# EPICS substitutions: iocBoot/iocgalil/galil_digital_ports.substitutions
# Description:
# digital/binary port substitution file.
#
# This library is free software; you can redistribute it and/or
# modify it under the terms of the GNU Lesser General Public
# Licence as published by the Free Software Foundation; either
# version 2.1 of the Licence, or (at your option) any later version.
#
# This library is distributed in the hope that it will be useful,
# but WITHOUT ANY WARRANTY; without even the implied warranty of
# MERCHANTABILITY or FITNESS FOR A PARTICULAR PURPOSE.  See the GNU
# Lesser General Public Licence for more details.
#
# You should have received a copy of the GNU Lesser General Public
# Licence along with this library; if not, write to the Free Software
# Foundation, Inc., 51 Franklin St, Fifth Floor, Boston, MA 02110-1301 USA.
#
# Contact details:
# mark.clift@synchrotron.org.au
# 800 Blackburn Road, Clayton, Victoria 3168, Australia.
#

# P    - PV prefix
# R    - Record Name
# PORT - Asyn port name
# BYTE - Hardware byte to read
# MASK - Mask for this bit

# Digital IO naming
# $(P)$(R)<Byte or word num><Type Bo or Bi><Bit>

file "$(TOP)/db/galil_digital_in_bit.template"
{
pattern {P,      R,          PORT,  BYTE,  MASK,     ZNAM,  ONAM,  ZSV,        OSV         }

# DMC = Digital motor controller
# DMC binary inputs are organized in bytes
	{CEL:GALIL,  Galil0Bi0,  Galil, 0,     0x000001, "Off", "On",  "NO_ALARM", "NO_ALARM"  }
	{CEL:GALIL,  Galil0Bi1,  Galil, 0,     0x000002, "Off", "On",  "NO_ALARM", "NO_ALARM"  }
	{CEL:GALIL,  Galil0Bi2,  Galil, 0,     0x000004, "Off", "On",  "NO_ALARM", "NO_ALARM"  }
	{CEL:GALIL,  Galil0Bi3,  Galil, 0,     0x000008, "Off", "On",  "NO_ALARM", "NO_ALARM"  }
	{CEL:GALIL,  Galil0Bi4,  Galil, 0,     0x000010, "Off", "On",  "NO_ALARM", "NO_ALARM"  }
	{CEL:GALIL,  Galil0Bi5,  Galil, 0,     0x000020, "Off", "On",  "NO_ALARM", "NO_ALARM"  }
	{CEL:GALIL,  Galil0Bi6,  Galil, 0,     0x000040, "Off", "On",  "NO_ALARM", "NO_ALARM"  }
	{CEL:GALIL,  Galil0Bi7,  Galil, 0,     0x000080, "Off", "On",  "NO_ALARM", "NO_ALARM"  }

	{CEL:GALIL,  Galil1Bi0,  Galil, 1,     0x000001, "Off", "On",  "NO_ALARM", "NO_ALARM"  }
	{CEL:GALIL,  Galil1Bi1,  Galil, 1,     0x000002, "Off", "On",  "NO_ALARM", "NO_ALARM"  }
	{CEL:GALIL,  Galil1Bi2,  Galil, 1,     0x000004, "Off", "On",  "NO_ALARM", "NO_ALARM"  }
	{CEL:GALIL,  Galil1Bi3,  Galil, 1,     0x000008, "Off", "On",  "NO_ALARM", "NO_ALARM"  }
	{CEL:GALIL,  Galil1Bi4,  Galil, 1,     0x000010, "Off", "On",  "NO_ALARM", "NO_ALARM"  }
	{CEL:GALIL,  Galil1Bi5,  Galil, 1,     0x000020, "Off", "On",  "NO_ALARM", "NO_ALARM"  }
	{CEL:GALIL,  Galil1Bi6,  Galil, 1,     0x000040, "Off", "On",  "NO_ALARM", "NO_ALARM"  }
	{CEL:GALIL,  Galil1Bi7,  Galil, 1,     0x000080, "Off", "On",  "NO_ALARM", "NO_ALARM"  }

	{CEL:GALIL,  Galil2Bi0,  Galil, 2,     0x000001, "Off", "On",  "NO_ALARM", "NO_ALARM"  }
	{CEL:GALIL,  Galil2Bi1,  Galil, 2,     0x000002, "Off", "On",  "NO_ALARM", "NO_ALARM"  }
	{CEL:GALIL,  Galil2Bi2,  Galil, 2,     0x000004, "Off", "On",  "NO_ALARM", "NO_ALARM"  }
	{CEL:GALIL,  Galil2Bi3,  Galil, 2,     0x000008, "Off", "On",  "NO_ALARM", "NO_ALARM"  }
	{CEL:GALIL,  Galil2Bi4,  Galil, 2,     0x000010, "Off", "On",  "NO_ALARM", "NO_ALARM"  }
	{CEL:GALIL,  Galil2Bi5,  Galil, 2,     0x000020, "Off", "On",  "NO_ALARM", "NO_ALARM"  }
	{CEL:GALIL,  Galil2Bi6,  Galil, 2,     0x000040, "Off", "On",  "NO_ALARM", "NO_ALARM"  }
	{CEL:GALIL,  Galil2Bi7,  Galil, 2,     0x000080, "Off", "On",  "NO_ALARM", "NO_ALARM"  }

# RIO binary inputs are organized in bytes
	{RIO01,  Galil0Bi0,  RIO,   0,     0x000001, "Off", "On",  "NO_ALARM", "NO_ALARM"  }
	{RIO01,  Galil0Bi1,  RIO,   0,     0x000002, "Off", "On",  "NO_ALARM", "NO_ALARM"  }
	{RIO01,  Galil0Bi2,  RIO,   0,     0x000004, "Off", "On",  "NO_ALARM", "NO_ALARM"  }
	{RIO01,  Galil0Bi3,  RIO,   0,     0x000008, "Off", "On",  "NO_ALARM", "NO_ALARM"  }
	{RIO01,  Galil0Bi4,  RIO,   0,     0x000010, "Off", "On",  "NO_ALARM", "NO_ALARM"  }
	{RIO01,  Galil0Bi5,  RIO,   0,     0x000020, "Off", "On",  "NO_ALARM", "NO_ALARM"  }
	{RIO01,  Galil0Bi6,  RIO,   0,     0x000040, "Off", "On",  "NO_ALARM", "NO_ALARM"  }
	{RIO01,  Galil0Bi7,  RIO,   0,     0x000080, "Off", "On",  "NO_ALARM", "NO_ALARM"  }

	{RIO01,  Galil1Bi0,  RIO,   1,     0x000001, "Off", "On",  "NO_ALARM", "NO_ALARM"  }
	{RIO01,  Galil1Bi1,  RIO,   1,     0x000002, "Off", "On",  "NO_ALARM", "NO_ALARM"  }
	{RIO01,  Galil1Bi2,  RIO,   1,     0x000004, "Off", "On",  "NO_ALARM", "NO_ALARM"  }
	{RIO01,  Galil1Bi3,  RIO,   1,     0x000008, "Off", "On",  "NO_ALARM", "NO_ALARM"  }
	{RIO01,  Galil1Bi4,  RIO,   1,     0x000010, "Off", "On",  "NO_ALARM", "NO_ALARM"  }
	{RIO01,  Galil1Bi5,  RIO,   1,     0x000020, "Off", "On",  "NO_ALARM", "NO_ALARM"  }
	{RIO01,  Galil1Bi6,  RIO,   1,     0x000040, "Off", "On",  "NO_ALARM", "NO_ALARM"  }
	{RIO01,  Galil1Bi7,  RIO,   1,     0x000080, "Off", "On",  "NO_ALARM", "NO_ALARM"  }

	{RIO01,  Galil2Bi0,  RIO,   2,     0x000001, "Off", "On",  "NO_ALARM", "NO_ALARM"  }
	{RIO01,  Galil2Bi1,  RIO,   2,     0x000002, "Off", "On",  "NO_ALARM", "NO_ALARM"  }
	{RIO01,  Galil2Bi2,  RIO,   2,     0x000004, "Off", "On",  "NO_ALARM", "NO_ALARM"  }
	{RIO01,  Galil2Bi3,  RIO,   2,     0x000008, "Off", "On",  "NO_ALARM", "NO_ALARM"  }
	{RIO01,  Galil2Bi4,  RIO,   2,     0x000010, "Off", "On",  "NO_ALARM", "NO_ALARM"  }
	{RIO01,  Galil2Bi5,  RIO,   2,     0x000020, "Off", "On",  "NO_ALARM", "NO_ALARM"  }
	{RIO01,  Galil2Bi6,  RIO,   2,     0x000040, "Off", "On",  "NO_ALARM", "NO_ALARM"  }
	{RIO01,  Galil2Bi7,  RIO,   2,     0x000080, "Off", "On",  "NO_ALARM", "NO_ALARM"  }

}

# P    - PV prefix
# R    - Record Name
# PORT - Asyn port name
# WORD - Hardware word to read
# MASK - Mask for this bit

file "$(TOP)/db/galil_digital_out_bit.template"
{
pattern {P,      R,           PORT,  WORD,  MASK,     ZNAM,  ONAM,  ZSV,        OSV         }

# DMC binary outputs are organized in 16bit words
	{CEL:GALIL,  Galil0Bo0,   Galil, 0,     0x000001, "Off", "On",  "NO_ALARM", "NO_ALARM"  }
	{CEL:GALIL,  Galil0Bo1,   Galil, 0,     0x000002, "Off", "On",  "NO_ALARM", "NO_ALARM"  }
	{CEL:GALIL,  Galil0Bo2,   Galil, 0,     0x000004, "Off", "On",  "NO_ALARM", "NO_ALARM"  }
	{CEL:GALIL,  Galil0Bo3,   Galil, 0,     0x000008, "Off", "On",  "NO_ALARM", "NO_ALARM"  }
	{CEL:GALIL,  Galil0Bo4,   Galil, 0,     0x000010, "Off", "On",  "NO_ALARM", "NO_ALARM"  }
	{CEL:GALIL,  Galil0Bo5,   Galil, 0,     0x000020, "Off", "On",  "NO_ALARM", "NO_ALARM"  }
	{CEL:GALIL,  Galil0Bo6,   Galil, 0,     0x000040, "Off", "On",  "NO_ALARM", "NO_ALARM"  }
	{CEL:GALIL,  Galil0Bo7,   Galil, 0,     0x000080, "Off", "On",  "NO_ALARM", "NO_ALARM"  }
	{CEL:GALIL,  Galil0Bo8,   Galil, 0,     0x000100, "Off", "On",  "NO_ALARM", "NO_ALARM"  }
	{CEL:GALIL,  Galil0Bo9,   Galil, 0,     0x000200, "Off", "On",  "NO_ALARM", "NO_ALARM"  }
	{CEL:GALIL,  Galil0Bo10,  Galil, 0,     0x000400, "Off", "On",  "NO_ALARM", "NO_ALARM"  }
	{CEL:GALIL,  Galil0Bo11,  Galil, 0,     0x000800, "Off", "On",  "NO_ALARM", "NO_ALARM"  }
	{CEL:GALIL,  Galil0Bo12,  Galil, 0,     0x001000, "Off", "On",  "NO_ALARM", "NO_ALARM"  }
	{CEL:GALIL,  Galil0Bo13,  Galil, 0,     0x002000, "Off", "On",  "NO_ALARM", "NO_ALARM"  }
	{CEL:GALIL,  Galil0Bo14,  Galil, 0,     0x004000, "Off", "On",  "NO_ALARM", "NO_ALARM"  }
	{CEL:GALIL,  Galil0Bo15,  Galil, 0,     0x008000, "Off", "On",  "NO_ALARM", "NO_ALARM"  }

	{CEL:GALIL,  Galil1Bo0,   Galil, 1,     0x000001, "Off", "On",  "NO_ALARM", "NO_ALARM"  }
	{CEL:GALIL,  Galil1Bo1,   Galil, 1,     0x000002, "Off", "On",  "NO_ALARM", "NO_ALARM"  }
	{CEL:GALIL,  Galil1Bo2,   Galil, 1,     0x000004, "Off", "On",  "NO_ALARM", "NO_ALARM"  }
	{CEL:GALIL,  Galil1Bo3,   Galil, 1,     0x000008, "Off", "On",  "NO_ALARM", "NO_ALARM"  }
	{CEL:GALIL,  Galil1Bo4,   Galil, 1,     0x000010, "Off", "On",  "NO_ALARM", "NO_ALARM"  }
	{CEL:GALIL,  Galil1Bo5,   Galil, 1,     0x000020, "Off", "On",  "NO_ALARM", "NO_ALARM"  }
	{CEL:GALIL,  Galil1Bo6,   Galil, 1,     0x000040, "Off", "On",  "NO_ALARM", "NO_ALARM"  }
	{CEL:GALIL,  Galil1Bo7,   Galil, 1,     0x000080, "Off", "On",  "NO_ALARM", "NO_ALARM"  }
	{CEL:GALIL,  Galil1Bo8,   Galil, 1,     0x000100, "Off", "On",  "NO_ALARM", "NO_ALARM"  }
	{CEL:GALIL,  Galil1Bo9,   Galil, 1,     0x000200, "Off", "On",  "NO_ALARM", "NO_ALARM"  }
	{CEL:GALIL,  Galil1Bo10,  Galil, 1,     0x000400, "Off", "On",  "NO_ALARM", "NO_ALARM"  }
	{CEL:GALIL,  Galil1Bo11,  Galil, 1,     0x000800, "Off", "On",  "NO_ALARM", "NO_ALARM"  }
	{CEL:GALIL,  Galil1Bo12,  Galil, 1,     0x001000, "Off", "On",  "NO_ALARM", "NO_ALARM"  }
	{CEL:GALIL,  Galil1Bo13,  Galil, 1,     0x002000, "Off", "On",  "NO_ALARM", "NO_ALARM"  }
	{CEL:GALIL,  Galil1Bo14,  Galil, 1,     0x004000, "Off", "On",  "NO_ALARM", "NO_ALARM"  }
	{CEL:GALIL,  Galil1Bo15,  Galil, 1,     0x008000, "Off", "On",  "NO_ALARM", "NO_ALARM"  }

# RIO binary outputs are organized in bytes
# However we name records in words for consistency with DMC for display purposes
	{RIO01,  Galil0Bo0,   RIO,   0,     0x000001, "Off", "On",  "NO_ALARM", "NO_ALARM"  }
	{RIO01,  Galil0Bo1,   RIO,   0,     0x000002, "Off", "On",  "NO_ALARM", "NO_ALARM"  }
	{RIO01,  Galil0Bo2,   RIO,   0,     0x000004, "Off", "On",  "NO_ALARM", "NO_ALARM"  }
	{RIO01,  Galil0Bo3,   RIO,   0,     0x000008, "Off", "On",  "NO_ALARM", "NO_ALARM"  }
	{RIO01,  Galil0Bo4,   RIO,   0,     0x000010, "Off", "On",  "NO_ALARM", "NO_ALARM"  }
	{RIO01,  Galil0Bo5,   RIO,   0,     0x000020, "Off", "On",  "NO_ALARM", "NO_ALARM"  }
	{RIO01,  Galil0Bo6,   RIO,   0,     0x000040, "Off", "On",  "NO_ALARM", "NO_ALARM"  }
	{RIO01,  Galil0Bo7,   RIO,   0,     0x000080, "Off", "On",  "NO_ALARM", "NO_ALARM"  }

	{RIO01,  Galil0Bo8,   RIO,   1,     0x000001, "Off", "On",  "NO_ALARM", "NO_ALARM"  }
	{RIO01,  Galil0Bo9,   RIO,   1,     0x000002, "Off", "On",  "NO_ALARM", "NO_ALARM"  }
	{RIO01,  Galil0Bo10,  RIO,   1,     0x000004, "Off", "On",  "NO_ALARM", "NO_ALARM"  }
	{RIO01,  Galil0Bo11,  RIO,   1,     0x000008, "Off", "On",  "NO_ALARM", "NO_ALARM"  }
	{RIO01,  Galil0Bo12,  RIO,   1,     0x000010, "Off", "On",  "NO_ALARM", "NO_ALARM"  }
	{RIO01,  Galil0Bo13,  RIO,   1,     0x000020, "Off", "On",  "NO_ALARM", "NO_ALARM"  }
	{RIO01,  Galil0Bo14,  RIO,   1,     0x000040, "Off", "On",  "NO_ALARM", "NO_ALARM"  }
	{RIO01,  Galil0Bo15,  RIO,   1,     0x000080, "Off", "On",  "NO_ALARM", "NO_ALARM"  }

	{RIO01,  Galil1Bo0,   RIO,   2,     0x000001, "Off", "On",  "NO_ALARM", "NO_ALARM"  }
	{RIO01,  Galil1Bo1,   RIO,   2,     0x000002, "Off", "On",  "NO_ALARM", "NO_ALARM"  }
	{RIO01,  Galil1Bo2,   RIO,   2,     0x000004, "Off", "On",  "NO_ALARM", "NO_ALARM"  }
	{RIO01,  Galil1Bo3,   RIO,   2,     0x000008, "Off", "On",  "NO_ALARM", "NO_ALARM"  }
	{RIO01,  Galil1Bo4,   RIO,   2,     0x000010, "Off", "On",  "NO_ALARM", "NO_ALARM"  }
	{RIO01,  Galil1Bo5,   RIO,   2,     0x000020, "Off", "On",  "NO_ALARM", "NO_ALARM"  }
	{RIO01,  Galil1Bo6,   RIO,   2,     0x000040, "Off", "On",  "NO_ALARM", "NO_ALARM"  }
	{RIO01,  Galil1Bo7,   RIO,   2,     0x000080, "Off", "On",  "NO_ALARM", "NO_ALARM"  }

}

# end
